{attribute 'qualified_only'}
VAR_GLOBAL
	dummyReporter:		FB_DummyDataReporter;
	defaultReporter:	I_DataReporter;
END_VAR

(* stored: Version 1.1.0.1, ProductVersion 3.1.4026.18
   GVL DATA_REPORTER_BASE: Id {1c3336c3-5d11-44c6-b11b-98725bf860ba} *)
